Fanuc KAREL source: kb00162.KL

-- PROVISIONAL review KL for V940-1; original PC SHA256 23c727d81c197e71dd6c6ce7821cecc0991848fa8786574ab65af0672060207d
-- Incomplete behavior may be omitted. Consult companion uncertainty JSON. Do not deploy.
PROGRAM KB00162
%NOLOCKGROUP
BEGIN
  -- V9_ZERO_TABLE_METADATA_HINT layout=0002_ascii; no indexed target words; source/name/runtime held
  -- UNRESOLVED_PC offsets 5-12; opcodes 9D,23
  -- UNRESOLVED_PC offsets 17-24; opcodes 9D,23
  -- UNRESOLVED_PC offsets 29-36; opcodes 9D,23
  -- UNRESOLVED_PC offsets 41-77; opcodes 27,22,22,22,1C,22,27,9D,31
  -- UNRESOLVED_PC offsets 82-86; opcodes 7F
END KB00162
